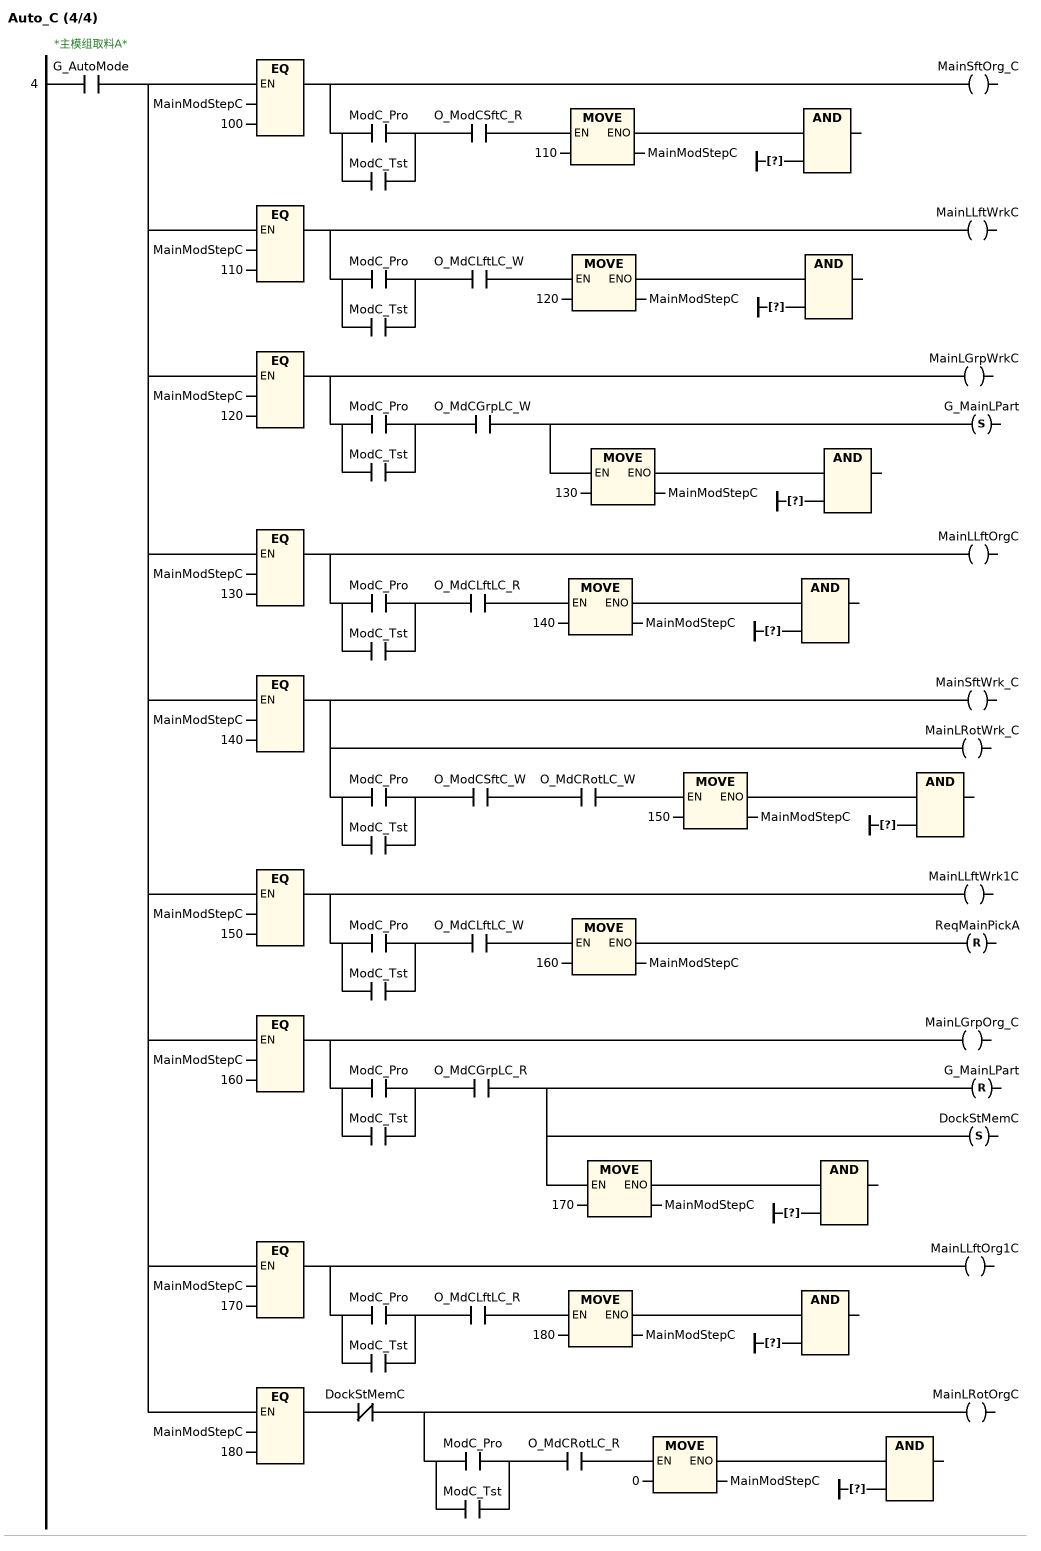
// NETWORK 4
// *主模组取料A*
_w22 := G_AutoMode AND MainModStepC = 100;
MainSftOrg_C := _w22;
_w23 := (_w22 AND ModC_Pro OR _w22 AND ModC_Tst) AND O_ModCSftC_R;
IF _w23 THEN MainModStepC := 110; END_IF
_w24 := G_AutoMode AND MainModStepC = 110;
MainLLftWrkC := _w24;
_w25 := (_w24 AND ModC_Pro OR _w24 AND ModC_Tst) AND O_MdCLftLC_W;
IF _w25 THEN MainModStepC := 120; END_IF
_w26 := G_AutoMode AND MainModStepC = 120;
MainLGrpWrkC := _w26;
_w27 := (_w26 AND ModC_Pro OR _w26 AND ModC_Tst) AND O_MdCGrpLC_W;
G_MainLPart S= _w27;
IF _w27 THEN MainModStepC := 130; END_IF
_w28 := G_AutoMode AND MainModStepC = 130;
MainLLftOrgC := _w28;
_w29 := (_w28 AND ModC_Pro OR _w28 AND ModC_Tst) AND O_MdCLftLC_R;
IF _w29 THEN MainModStepC := 140; END_IF
_w30 := G_AutoMode AND MainModStepC = 140;
MainSftWrk_C := _w30;
MainLRotWrk_C := _w30;
_w31 := (_w30 AND ModC_Pro OR _w30 AND ModC_Tst) AND O_ModCSftC_W AND O_MdCRotLC_W;
IF _w31 THEN MainModStepC := 150; END_IF
_w32 := G_AutoMode AND MainModStepC = 150;
MainLLftWrk1C := _w32;
_w33 := (_w32 AND ModC_Pro OR _w32 AND ModC_Tst) AND O_MdCLftLC_W;
IF _w33 THEN MainModStepC := 160; END_IF
ReqMainPickA R= _w33;
_w34 := G_AutoMode AND MainModStepC = 160;
MainLGrpOrg_C := _w34;
_w35 := (_w34 AND ModC_Pro OR _w34 AND ModC_Tst) AND O_MdCGrpLC_R;
G_MainLPart R= _w35;
DockStMemC S= _w35;
IF _w35 THEN MainModStepC := 170; END_IF
_w36 := G_AutoMode AND MainModStepC = 170;
MainLLftOrg1C := _w36;
_w37 := (_w36 AND ModC_Pro OR _w36 AND ModC_Tst) AND O_MdCLftLC_R;
IF _w37 THEN MainModStepC := 180; END_IF
_w38 := (G_AutoMode AND MainModStepC = 180) AND NOT DockStMemC;
MainLRotOrgC := _w38;
_w39 := (_w38 AND ModC_Pro OR _w38 AND ModC_Tst) AND O_MdCRotLC_R;
IF _w39 THEN MainModStepC := 0; END_IF

END_PROGRAM

// Device/Application/03_程序/输出/Cylinder_AZone
PROGRAM Cylinder_AZone
VAR
	StopA1Hm :BOOL;
	StopA1Wk :BOOL;
	StopA2Hm :BOOL;
	StopA2Wk :BOOL;
	StopA3Hm :BOOL;
	StopA3Wk :BOOL;
	StopA4Hm :BOOL;
	StopA4Wk :BOOL;
	StopA5Hm :BOOL;
	StopA5Wk :BOOL;
	LiftA1Hm: BOOL;
	LiftA1Wk: BOOL ;
	LiftA2Hm: BOOL;
	LiftA2Wk: BOOL ;
	LiftA3Hm: BOOL;
	LiftA3Wk: BOOL ;
	LiftA4Hm: BOOL;
	LiftA4Wk: BOOL ;
	SwtchA1Hm: BOOL;
	SwtchA1Wk: BOOL ;
	ModTrvAHm: BOOL;
	ModTrvAWk: BOOL ;
	ModClpAHm: BOOL;
	ModClpAWk: BOOL; 
	ModRotAHm: BOOL;
	ModRotAWk: BOOL; 
	
	FB_StopA1: FB_Cylinder;
	FB_StopA2: FB_Cylinder;
	FB_StopA3: FB_Cylinder;
	FB_StopA4: FB_Cylinder;
	FB_StopA5: FB_Cylinder;
	FB_LiftA1: FB_Cylinder;
    FB_LiftA2: FB_Cylinder;
    FB_LiftA3: FB_Cylinder;
    FB_LiftA4: FB_Cylinder;
	FB_SwtchA1: FB_Cylinder;
	FB_ModTrvA: FB_Cylinder;
	FB_ModClpA: FB_Cylinder;
	FB_ModRotA: FB_Cylinder;
END_VAR

//阻挡气缸A1//
IF (G_ManMode AND H_StpC_R_A1) OR LnCylInit_A.Y_BlkCylR1 OR St1Org_A
THEN StopA1Hm:=TRUE;
ELSE StopA1Hm:=FALSE;
END_IF;
IF (G_ManMode AND H_StpC_W_A1) OR St1Work_A
THEN StopA1Wk:=TRUE;
ELSE StopA1Wk:=FALSE;
END_IF;
FB_StopA1(
 X_EN:=1,
 X_HomeInBit:=X_StpCyl_R_A1,
 X_WorkInBit:=X_StpCyl_W_A1,
 X_HomeCmdBit:=StopA1Hm,
 X_WorkCmdBit:=StopA1Wk,
 X_HomeMskBit:=H_StpCR_A1_M,
 X_WorkMskBit:=H_StpCW_A1_M,
 X_HomeConfT:=H_StpCRPosDyA1,
 X_WorkConfT:=H_StpCWPosDyA1,
 X_TimeoutSet:=H_StpCTO_DlyA1,
 X_HomeMskDly:=H_StpCRMaskDyA1,
 X_WorkMskDly:=H_StpCWMaskDyA1,
 Y_ENO=>,
 Y_AtHome=>O_StpC_R_A1,
 Y_AtWork=>O_StpC_W_A1,
 Y_HomeTout=>O_StpCRFltA1,
 Y_WorkTout=>O_StpCRFltA1,
 Y_HomeOutBit=>Q_StpCyl_R_A1,
 Y_WorkOutBit=>Q_StpCyl_W_A1);
//阻挡气缸A2//
IF (G_ManMode AND H_StpC_R_A2) OR LnCylInit_A.Y_BlkCylR2 OR St2Org_A
THEN StopA2Hm:=TRUE;
ELSE StopA2Hm:=FALSE;
END_IF;
IF (G_ManMode AND H_StpC_W_A2)  OR St2Work_A
THEN StopA2Wk:=TRUE;
ELSE StopA2Wk:=FALSE;
END_IF;
FB_StopA2(
 X_EN:=1,
 X_HomeInBit:=X_StpCyl_R_A2,
 X_WorkInBit:=X_StpCyl_W_A2,
 X_HomeCmdBit:=StopA2Hm,
 X_WorkCmdBit:=StopA2Wk,
 X_HomeMskBit:=H_StpCR_A2_M,
 X_WorkMskBit:=H_StpCW_A2_M,
 X_HomeConfT:=H_StpCRPosDyA2,
 X_WorkConfT:=H_StpCWPosDyA2,
 X_TimeoutSet:=H_StpCTO_DlyA2,
 X_HomeMskDly:=H_StpCRMaskDyA2,
 X_WorkMskDly:=H_StpCWMaskDyA2,
 Y_ENO=>,
 Y_AtHome=>O_StpC_R_A2,
 Y_AtWork=>O_StpC_W_A2,
 Y_HomeTout=>O_StpCRFltA2,
 Y_WorkTout=>O_StpCWFltA2,
 Y_HomeOutBit=>Q_StpCyl_R_A2,
 Y_WorkOutBit=>Q_StpCyl_W_A2);
//阻挡气缸A3//
IF (G_ManMode AND H_StpC_R_A3) OR LnCylInit_A.Y_BlkCylR3 OR St3Org_A
THEN StopA3Hm:=TRUE;
ELSE StopA3Hm:=FALSE;
END_IF;
IF (G_ManMode AND H_StpC_W_A3)  OR St3Work_A OR St3Work1_A
THEN StopA3Wk:=TRUE;
ELSE StopA3Wk:=FALSE;
END_IF;
FB_StopA3(
 X_EN:=1,
 X_HomeInBit:=X_StpCyl_R_A3,
 X_WorkInBit:=X_StpCyl_W_A3,
 X_HomeCmdBit:=StopA3Hm,
 X_WorkCmdBit:=StopA3Wk,
 X_HomeMskBit:=H_StpCR_A3_M,
 X_WorkMskBit:=H_StpCW_A3_M,
 X_HomeConfT:=H_StpCRPosDyA3,
 X_WorkConfT:=H_StpCWPosDyA3,
 X_TimeoutSet:=H_StpCTO_DlyA3,
 X_HomeMskDly:=H_StpCRMaskDyA3,
 X_WorkMskDly:=H_StpCWMaskDyA3,
 Y_ENO=>,
 Y_AtHome=>O_StpC_R_A3,
 Y_AtWork=>O_StpC_W_A3,
 Y_HomeTout=>O_StpCRFltA3,
 Y_WorkTout=>O_StpCWFltA3,
 Y_HomeOutBit=>Q_StpCyl_R_A3,
 Y_WorkOutBit=>Q_StpCyl_W_A3);
//阻挡气缸A4//
IF (G_ManMode AND H_StpC_R_A4) OR LnCylInit_A.Y_BlkCylR4 OR St4Org_A
THEN StopA4Hm:=TRUE;
ELSE StopA4Hm:=FALSE;
END_IF;
IF (G_ManMode AND H_StpC_W_A4)  OR St4Work_A
THEN StopA4Wk:=TRUE;
ELSE StopA4Wk:=FALSE;
END_IF;
FB_StopA4(
 X_EN:=1,
 X_HomeInBit:=X_StpCyl_R_A4,
 X_WorkInBit:=X_StpCyl_W_A4,
 X_HomeCmdBit:=StopA4Hm,
 X_WorkCmdBit:=StopA4Wk,
 X_HomeMskBit:=H_StpCR_A4_M,
 X_WorkMskBit:=H_StpCW_A4_M,
 X_HomeConfT:=H_StpCRPosDyA4,
 X_WorkConfT:=H_StpCWPosDyA4,
 X_TimeoutSet:=H_StpCTO_DlyA4,
 X_HomeMskDly:=H_StpCRMaskDyA4,
 X_WorkMskDly:=H_StpCWMaskDyA4,
 Y_ENO=>,
 Y_AtHome=>O_StpC_R_A4,
 Y_AtWork=>O_StpC_W_A4,
 Y_HomeTout=>O_StpCRFltA4,
 Y_WorkTout=>O_StpCWFltA4,
 Y_HomeOutBit=>Q_StpCyl_R_A4,
 Y_WorkOutBit=>Q_StpCyl_W_A4);
//阻挡气缸A5//
IF (G_ManMode AND H_StpC_R_A5) OR LnCylInit_A.Y_BlkCylR5 OR St5Org_A
THEN StopA5Hm:=TRUE;
ELSE StopA5Hm:=FALSE;
END_IF;
IF (G_ManMode AND H_StpC_W_A5) OR St5Work_A
THEN StopA5Wk:=TRUE;
ELSE StopA5Wk:=FALSE;
END_IF;
FB_StopA5(
 X_EN:=1,
 X_HomeInBit:=X_StpCyl_R_A5,
 X_WorkInBit:=X_StpCyl_W_A5,
 X_HomeCmdBit:=StopA5Hm,
 X_WorkCmdBit:=StopA5Wk,
 X_HomeMskBit:=H_StpCR_A5_M,
 X_WorkMskBit:=H_StpCW_A5_M,
 X_HomeConfT:=H_StpCRPosDyA5,
 X_WorkConfT:=H_StpCWPosDyA5,
 X_TimeoutSet:=H_StpCTO_DlyA5,
 X_HomeMskDly:=H_StpCRMaskDyA5,
 X_WorkMskDly:=H_StpCWMaskDyA5,
 Y_ENO=>,
 Y_AtHome=>O_StpC_R_A5,
 Y_AtWork=>O_StpC_W_A5,
 Y_HomeTout=>O_StpCRFltA5,
 Y_WorkTout=>O_StpCWFltA5,
 Y_HomeOutBit=>Q_StpCyl_R_A5,
 Y_WorkOutBit=>Q_StpCyl_W_A5);
//顶升气缸A1//
IF (G_ManMode AND H_LftC_R_A1) OR LnCylInit_A.Y_LftCylR1 OR UD1Org_A OR UD1OrgPos1_A
THEN LiftA1Hm:=TRUE;
ELSE LiftA1Hm:=FALSE;
END_IF;
IF (G_ManMode AND H_LftC_W_A1) OR LnCylInit_A.Y_LftCylM1 OR UD1Work_A OR UD1Work1_A
THEN LiftA1Wk:=TRUE;
ELSE LiftA1Wk:=FALSE;
END_IF;
FB_LiftA1(
 X_EN:=1,
 X_HomeInBit:=X_LftCyl_R_A1,
 X_WorkInBit:=X_LftCyl_W_A1,
 X_HomeCmdBit:=LiftA1Hm,
 X_WorkCmdBit:=LiftA1Wk,
 X_HomeMskBit:=H_LftCR_A1_M,
 X_WorkMskBit:=H_LftCW_A1_M,
 X_HomeConfT:=H_LftCRPosDyA1,
 X_WorkConfT:=H_LftCWPosDyA1,
 X_TimeoutSet:=H_LftCTO_DlyA1,
 X_HomeMskDly:=H_LftCRMaskDyA1,
 X_WorkMskDly:=H_LftCWMaskDyA1,
 Y_ENO=>,
 Y_AtHome=>O_LftC_R_A1,
 Y_AtWork=>O_LftC_W_A1,
 Y_HomeTout=>O_LftCRFltA1,
 Y_WorkTout=>O_LftCWFltA1,
 Y_HomeOutBit=>Q_LftCyl_R_A1,
 Y_WorkOutBit=>Q_LftCyl_W_A1);
//顶升气缸A2//
IF (G_ManMode AND H_LftC_R_A2) OR LnCylInit_A.Y_LftCylR2 OR UD2Org_A
THEN LiftA2Hm:=TRUE;
ELSE LiftA2Hm:=FALSE;
END_IF;
IF (G_ManMode AND H_LftC_W_A2)  OR UD2Work_A
THEN LiftA2Wk:=TRUE;
ELSE LiftA2Wk:=FALSE;
END_IF;
FB_LiftA2(
 X_EN:=1,
 X_HomeInBit:=X_LftCyl_R_A2,
 X_WorkInBit:=X_LftCyl_W_A2,
 X_HomeCmdBit:=LiftA2Hm,
 X_WorkCmdBit:=LiftA2Wk,
 X_HomeMskBit:=H_LftCR_A2_M,
 X_WorkMskBit:=H_LftCW_A2_M,
 X_HomeConfT:=H_LftCRPosDyA2,
 X_WorkConfT:=H_LftCWPosDyA2,
 X_TimeoutSet:=H_LftCTO_DlyA2,
 X_HomeMskDly:=H_LftCRMaskDyA2,
 X_WorkMskDly:=H_LftCWMaskDyA2,
 Y_ENO=>,
 Y_AtHome=>O_LftC_R_A2,
 Y_AtWork=>O_LftC_W_A2,
 Y_HomeTout=>O_LftCRFltA2,
 Y_WorkTout=>O_LftCWFltA2,
 Y_HomeOutBit=>Q_LftCyl_R_A2,
 Y_WorkOutBit=>Q_LftCyl_W_A2);
//顶升气缸A3//
IF (G_ManMode AND H_LftC_R_A3) OR LnCylInit_A.Y_LftCylR3 OR UD3Org_A
THEN LiftA3Hm:=TRUE;
ELSE LiftA3Hm:=FALSE;
END_IF;
IF (G_ManMode AND H_LftC_W_A3)  OR UD3Work_A
THEN LiftA3Wk:=TRUE;
ELSE LiftA3Wk:=FALSE;
END_IF;
FB_LiftA3(
 X_EN:=1,
 X_HomeInBit:=X_LftCyl_R_A3,
 X_WorkInBit:=X_LftCyl_W_A3,
 X_HomeCmdBit:=LiftA3Hm,
 X_WorkCmdBit:=LiftA3Wk,
 X_HomeMskBit:=H_LftCR_A3_M,
 X_WorkMskBit:=H_LftCW_A3_M,
 X_HomeConfT:=H_LftCRPosDyA3,
 X_WorkConfT:=H_LftCWPosDyA3,
 X_TimeoutSet:=H_LftCTO_DlyA3,
 X_HomeMskDly:=H_LftCRMaskDyA3,
 X_WorkMskDly:=H_LftCWMaskDyA3,
 Y_ENO=>,
 Y_AtHome=>O_LftC_R_A3,
 Y_AtWork=>O_LftC_W_A3,
 Y_HomeTout=>O_LftCRFltA3,
 Y_WorkTout=>O_LftCWFltA3,
 Y_HomeOutBit=>Q_LftCyl_R_A3,
 Y_WorkOutBit=>Q_LftCyl_W_A3);
//顶升气缸A4//
IF (G_ManMode AND H_LftC_R_A4) OR LnCylInit_A.Y_LftCylR4 OR UD4Org_A
THEN LiftA4Hm:=TRUE;
ELSE LiftA4Hm:=FALSE;
END_IF;
IF (G_ManMode AND H_LftC_W_A4)  OR UD4Work_A
THEN LiftA4Wk:=TRUE;
ELSE LiftA4Wk:=FALSE;
END_IF;
FB_LiftA4(
 X_EN:=1,
 X_HomeInBit:=X_LftCyl_R_A4,
 X_WorkInBit:=X_LftCyl_W_A4,
 X_HomeCmdBit:=LiftA4Hm,
 X_WorkCmdBit:=LiftA4Wk,
 X_HomeMskBit:=H_LftCR_A4_M,
 X_WorkMskBit:=H_LftCW_A4_M,
 X_HomeConfT:=H_LftCRPosDyA4,
 X_WorkConfT:=H_LftCWPosDyA4,
 X_TimeoutSet:=H_LftCTO_DlyA4,
 X_HomeMskDly:=H_LftCRMaskDyA4,
 X_WorkMskDly:=H_LftCWMaskDyA4,
 Y_ENO=>,
 Y_AtHome=>O_LftC_R_A4,
 Y_AtWork=>O_LftC_W_A4,
 Y_HomeTout=>O_LftCRFltA4,
 Y_WorkTout=>O_LftCWFltA4,
 Y_HomeOutBit=>Q_LftCyl_R_A4,
 Y_WorkOutBit=>Q_LftCyl_W_A4);
//换向气缸A1//
IF (G_ManMode AND H_TrnC_R_A1 AND O_LftC_W_A1) OR LnCylInit_A.Y_StrCylO1 OR RevOrg_A
THEN SwtchA1Hm:=TRUE;
ELSE SwtchA1Hm:=FALSE;
END_IF;
IF (G_ManMode AND H_TrnC_W_A1 AND O_LftC_W_A1)  OR RevWork_A
THEN SwtchA1Wk:=TRUE;
ELSE SwtchA1Wk:=FALSE;
END_IF;
FB_SwtchA1(
 X_EN:=1,
 X_HomeInBit:=X_TrnCyl_R_A1,
 X_WorkInBit:=X_TrnCyl_W_A1,
 X_HomeCmdBit:=SwtchA1Hm,
 X_WorkCmdBit:=SwtchA1Wk,
 X_HomeMskBit:=H_TrnCR_A1_M,
 X_WorkMskBit:=H_TrnCW_A1_M ,
 X_HomeConfT:=H_TrnCRPosDyA1,
 X_WorkConfT:=H_TrnCWPosDyA1,
 X_TimeoutSet:=H_TrnCTO_DlyA1,
 X_HomeMskDly:=H_TrnCRMaskDyA1,
 X_WorkMskDly:=H_TrnCWMaskDyA1,
 Y_ENO=>,
 Y_AtHome=>O_TrnC_R_A1,
 Y_AtWork=>O_TrnC_W_A1,
 Y_HomeTout=>O_TrnCRFltA1,
 Y_WorkTout=>O_TrnCWFltA1,
 Y_HomeOutBit=>Q_TrnCyl_R_A1,
 Y_WorkOutBit=>Q_TrnCyl_W_A1);
//模组平移气缸A//
IF (G_ManMode AND H_ModASftC_R AND Ax1GoP1) OR PickModInitA.Y_TrnCylR OR SftCylOrg_A
THEN ModTrvAHm:=TRUE;
ELSE ModTrvAHm:=FALSE;
END_IF;
IF (G_ManMode AND H_ModASftC_W AND Ax1GoP1)  OR SftCylWork_A
THEN ModTrvAWk:=TRUE;
ELSE ModTrvAWk:=FALSE;
END_IF;
FB_ModTrvA(
 X_EN:=1,
 X_HomeInBit:=X_ModASftC_R,
 X_WorkInBit:=X_ModASftC_W,
 X_HomeCmdBit:=ModTrvAHm,
 X_WorkCmdBit:=ModTrvAWk,
 X_HomeMskBit:=H_MdASftCR_M,
 X_WorkMskBit:=H_MdASftCW_M,
 X_HomeConfT:=H_MASftCRPosDy,
 X_WorkConfT:=H_MASftCWPosDy,
 X_TimeoutSet:=H_MASftCTO_Dly,
 X_HomeMskDly:=H_MASftCRMaskDy,
 X_WorkMskDly:=H_MASftCWMaskDy,
 Y_ENO=>,
 Y_AtHome=>O_ModASftC_R,
 Y_AtWork=>O_ModASftC_W,
 Y_HomeTout=>O_MASftCRFlt,
 Y_WorkTout=>O_MASftCWFlt,
 Y_HomeOutBit=>Q_ModASftC_R,
 Y_WorkOutBit=>Q_ModASftC_W);
//模组夹取气缸A//
IF (G_ManMode AND H_ModAGrpC_R) OR PickModInitA.Y_ClmpCylO OR GripCylOrg_A
THEN ModClpAHm:=TRUE;
ELSE ModClpAHm:=FALSE;
END_IF;
IF (G_ManMode AND H_ModAGrpC_W) OR GripCylWorkA
THEN ModClpAWk:=TRUE;
ELSE ModClpAWk:=FALSE;
END_IF;
FB_ModClpA(
 X_EN:=1,
 X_HomeInBit:=X_ModAGrpC_R,
 X_WorkInBit:=X_ModAGrpC_W,
 X_HomeCmdBit:=ModClpAHm,
 X_WorkCmdBit:=ModClpAWk,
 X_HomeMskBit:=H_MdAGrpCR_M,
 X_WorkMskBit:=H_MdAGrpCW_M,
 X_HomeConfT:=H_MAGrpCRPosDy,
 X_WorkConfT:=H_MAGrpCWPosDy,
 X_TimeoutSet:=H_MAGrpCTO_Dly,
 X_HomeMskDly:=H_MAGrpCRMaskDy,
 X_WorkMskDly:=H_MAGrpCWMaskDy,
 Y_ENO=>,
 Y_AtHome=>O_ModAGrpC_R,
 Y_AtWork=>O_ModAGrpC_W,
 Y_HomeTout=>O_MAGrpCRFlt,
 Y_WorkTout=>O_MAGrpCWFlt,
 Y_HomeOutBit=>Q_ModAGrpC_R,
 Y_WorkOutBit=>Q_ModAGrpC_W);
//模组旋转气缸A//
IF (G_ManMode AND H_ModARotC_R) OR PickModInitA.Y_RotCylO OR RotCylOrg_A
THEN ModRotAHm:=TRUE;
ELSE ModRotAHm:=FALSE;
END_IF;
IF (G_ManMode AND H_ModARotC_W) OR RotCylWork_A
THEN ModRotAWk:=TRUE;
ELSE ModRotAWk:=FALSE;
END_IF;
FB_ModRotA(
 X_EN:=1,
 X_HomeInBit:=X_ModARotC_R,
 X_WorkInBit:=X_ModARotC_W,
 X_HomeCmdBit:=ModRotAHm,
 X_WorkCmdBit:=ModRotAWk,
 X_HomeMskBit:=H_MdARotCR_M,
 X_WorkMskBit:=H_MdARotCW_M,
 X_HomeConfT:=H_MARotCRPosDy,
 X_WorkConfT:=H_MARotCWPosDy,
 X_TimeoutSet:=H_MARotCTO_Dly,
 X_HomeMskDly:=H_MARotCRMaskDy,
 X_WorkMskDly:=H_MARotCWMaskDy,
 Y_ENO=>,
 Y_AtHome=>O_ModARotC_R,
 Y_AtWork=>O_ModARotC_W,
 Y_HomeTout=>O_MARotCRFlt,
 Y_WorkTout=>O_MARotCWFlt,
 Y_HomeOutBit=>Q_ModARotC_R,
 Y_WorkOutBit=>Q_ModARotC_W);

END_PROGRAM

// Device/Application/02_功能块/气缸/FB_Cylinder
FUNCTION_BLOCK FB_Cylinder
VAR_INPUT
	X_EN: BOOL;
	X_HomeInBit: BOOL;
	X_WorkInBit: BOOL;
	X_HomeCmdBit: BOOL;
	X_WorkCmdBit: BOOL;
	X_HomeMskBit: BOOL;
	X_WorkMskBit: BOOL;
	X_HomeConfT: TIME;
	X_WorkConfT: TIME;
	X_TimeoutSet: TIME;
	X_HomeMskDly: TIME;
	X_WorkMskDly: TIME;
END_VAR
VAR_OUTPUT
	Y_ENO: BOOL;
	Y_AtHome: BOOL;
	Y_AtWork: BOOL;
	Y_HomeTout: BOOL;
	Y_WorkTout: BOOL;
	Y_HomeOutBit: BOOL;
	Y_WorkOutBit: BOOL;	
END_VAR
VAR
	TON_0: TON;
	TON_1: TON;
	TON_2: TON;
	TON_3: TON;
	TON_4: TON;
	TON_5: TON;
	R_TRIG_0: R_TRIG;
	END_VAR
VAR // added by the converter: edge detectors and wires of the graphical bodies
    _w1, _w2, _w3, _w4, _w5 : BOOL;
END_VAR

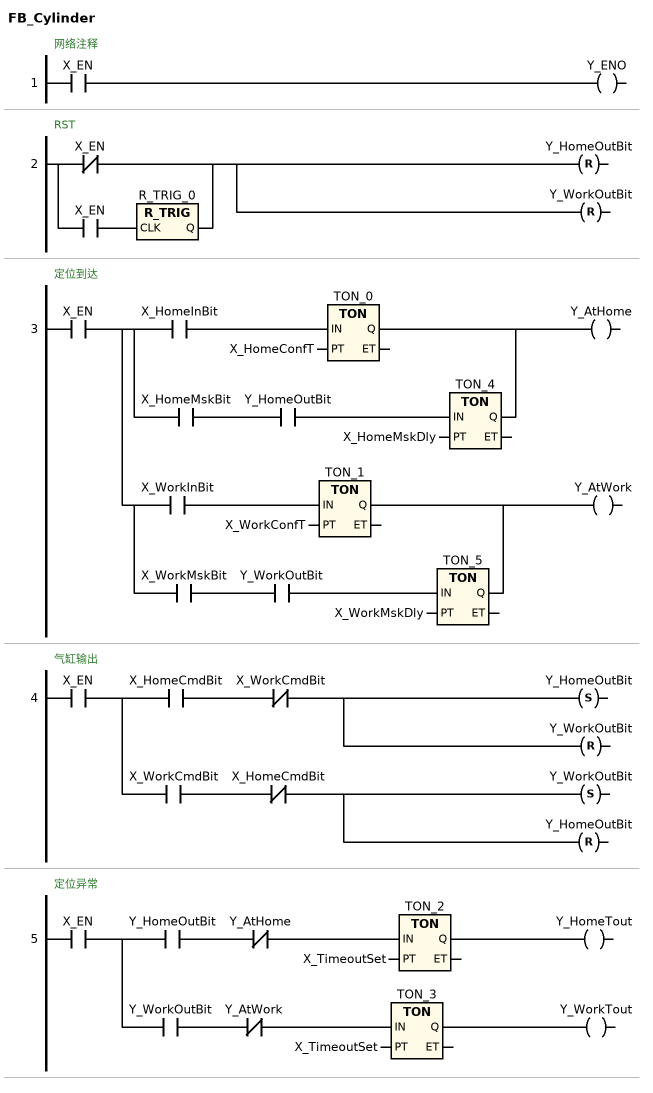
// NETWORK 1
// 网络注释
Y_ENO := X_EN;

// NETWORK 2
// RST
R_TRIG_0(CLK := X_EN); // R_TRIG
_w1 := NOT X_EN OR R_TRIG_0.Q;
Y_HomeOutBit R= _w1;
Y_WorkOutBit R= _w1;

// NETWORK 3
// 定位到达
TON_0(IN := X_EN AND X_HomeInBit, PT := X_HomeConfT); // TON
TON_4(IN := (X_EN AND X_HomeMskBit) AND Y_HomeOutBit, PT := X_HomeMskDly); // TON
_w2 := TON_0.Q OR TON_4.Q;
Y_AtHome := _w2;
TON_1(IN := X_EN AND X_WorkInBit, PT := X_WorkConfT); // TON
TON_5(IN := (X_EN AND X_WorkMskBit) AND Y_WorkOutBit, PT := X_WorkMskDly); // TON
_w3 := TON_1.Q OR TON_5.Q;
Y_AtWork := _w3;

// NETWORK 4
// 气缸输出
_w4 := (X_EN AND X_HomeCmdBit) AND NOT X_WorkCmdBit;
Y_HomeOutBit S= _w4;
Y_WorkOutBit R= _w4;
_w5 := (X_EN AND X_WorkCmdBit) AND NOT X_HomeCmdBit;
Y_WorkOutBit S= _w5;
Y_HomeOutBit R= _w5;

// NETWORK 5
// 定位异常
TON_2(IN := (X_EN AND Y_HomeOutBit) AND NOT Y_AtHome, PT := X_TimeoutSet); // TON
Y_HomeTout := TON_2.Q;
TON_3(IN := (X_EN AND Y_WorkOutBit) AND NOT Y_AtWork, PT := X_TimeoutSet); // TON
Y_WorkTout := TON_3.Q;

END_FUNCTION_BLOCK

// Device/Application/03_程序/输出/Cylinder_CZone
PROGRAM Cylinder_CZone
VAR
 StopC1Hm :BOOL;
 StopC1Wk :BOOL;
 LiftC1Hm: BOOL;
 LiftC1Wk: BOOL ;
ModTrvCHm :BOOL;
ModTrvCWk :BOOL;
ModLLftCHm :BOOL;
ModLLftCWk :BOOL;
ModLClpCHm :BOOL;
ModLClpCWk :BOOL;
ModLRotCHm :BOOL;
ModLRotCWk :BOOL;

 
 FB_StopC1: FB_Cylinder;
 FB_LiftC1: FB_Cylinder;
 FB_ModTrvC: FB_Cylinder;
 FB_ModLLftC: FB_Cylinder;
 FB_ModLClpC: FB_Cylinder;
 FB_ModLRotC: FB_Cylinder;
END_VAR

//阻挡气缸C1//
IF (G_ManMode AND H_StpC_R_C1) OR DockCylInitC.Y_BlkCylR OR StpCylOrg_C
THEN StopC1Hm:=TRUE;
ELSE StopC1Hm:=FALSE;
END_IF;
IF (G_ManMode AND H_StpC_W_C1) OR StpCylWork_C
THEN StopC1Wk:=TRUE;
ELSE StopC1Wk:=FALSE;
END_IF;
FB_StopC1(
 X_EN:=1,
 X_HomeInBit:=X_StpCyl_R_C1,
 X_WorkInBit:=X_StpCyl_W_C1,
 X_HomeCmdBit:=StopC1Hm,
 X_WorkCmdBit:=StopC1Wk,
 X_HomeMskBit:=H_StpCR_C1_M,
 X_WorkMskBit:=H_StpCW_C1_M,
 X_HomeConfT:=H_StpCRPosDyC1,
 X_WorkConfT:=H_StpCWPosDyC1,
 X_TimeoutSet:=H_StpCTO_DlyC1,
 X_HomeMskDly:=H_StpCRMaskDyC1,
 X_WorkMskDly:=H_StpCWMaskDyC1,
 Y_ENO=>,
 Y_AtHome=>O_StpC_R_C1,
 Y_AtWork=>O_StpC_W_C1,
 Y_HomeTout=>O_StpCRFltC1,
 Y_WorkTout=>O_StpCWFltC1,
 Y_HomeOutBit=>Q_StpCyl_R_C1,
 Y_WorkOutBit=>Q_StpCyl_W_C1);
//顶升气缸C1//
IF (G_ManMode AND H_LftC_R_C1) OR DockCylInitC.Y_LftCylR OR LftCylOrg_C
THEN LiftC1Hm:=TRUE;
ELSE LiftC1Hm:=FALSE;
END_IF;
IF (G_ManMode AND H_LftC_W_C1) OR LftCylWork_C
THEN LiftC1Wk:=TRUE;
ELSE LiftC1Wk:=FALSE;
END_IF;
FB_LiftC1(
 X_EN:=1,
 X_HomeInBit:=X_LftCyl_R_C1,
 X_WorkInBit:=X_LftCyl_W_C1,
 X_HomeCmdBit:=LiftC1Hm,
 X_WorkCmdBit:=LiftC1Wk,
 X_HomeMskBit:=H_LftCR_C1_M,
 X_WorkMskBit:=H_LftCW_C1_M,
 X_HomeConfT:=H_LftCRPosDyC1,
 X_WorkConfT:=H_LftCWPosDyC1,
 X_TimeoutSet:=H_LftCTO_DlyC1,
 X_HomeMskDly:=H_LftCRMaskDyC1,
 X_WorkMskDly:=H_LftCWMaskDyC1,
 Y_ENO=>,
 Y_AtHome=>O_LftC_R_C1,
 Y_AtWork=>O_LftC_W_C1,
 Y_HomeTout=>O_LftCRFltC1,
 Y_WorkTout=>O_LftCWFltC1,
 Y_HomeOutBit=>Q_LftCyl_R_C1,
 Y_WorkOutBit=>Q_LftCyl_W_C1);
//模组平移气缸C//
IF (G_ManMode AND H_ModCSftC_R AND O_MdCLftLC_R) OR MainModInitC.Y_TrnCylR OR MainSftOrg_C OR MainSftOrg1C
THEN ModTrvCHm:=TRUE;
ELSE ModTrvCHm:=FALSE;
END_IF;
IF (G_ManMode AND H_ModCSftC_W AND O_MdCLftLC_R)  OR MainSftWrk_C OR MainSftWrk1_C
THEN ModTrvCWk:=TRUE;
ELSE ModTrvCWk:=FALSE;
END_IF;
FB_ModTrvC(
 X_EN:=1,
 X_HomeInBit:=X_ModCSftC_R,
 X_WorkInBit:=X_ModCSftC_W,
 X_HomeCmdBit:=ModTrvCHm,
 X_WorkCmdBit:=ModTrvCWk,
 X_HomeMskBit:=H_MdCSftCR_M,
 X_WorkMskBit:=H_MdCSftCW_M,
 X_HomeConfT:=H_MCSftCRPosDy,
 X_WorkConfT:=H_MCSftCWPosDy,
 X_TimeoutSet:=H_MCSftCTO_Dly,
 X_HomeMskDly:=H_MCSftCRMaskDy,
 X_WorkMskDly:=H_MCSftCWMaskDy,
 Y_ENO=>,
 Y_AtHome=>O_ModCSftC_R,
 Y_AtWork=>O_ModCSftC_W,
 Y_HomeTout=>O_MCSftCRFlt,
 Y_WorkTout=>O_MCSftCWFlt,
 Y_HomeOutBit=>Q_ModCSftC_R,
 Y_WorkOutBit=>Q_ModCSftC_W);
//模组左升降气缸C//
IF (G_ManMode AND H_MdCLftLC_R) OR MainModInitC.Y_LLftCylR OR MainLLftOrgC OR MainLLftOrg1C
THEN ModLLftCHm:=TRUE;
ELSE ModLLftCHm:=FALSE;
END_IF;
IF (G_ManMode AND H_MdCLftLC_W)  OR MainLLftWrkC  OR MainLLftWrk1C
THEN ModLLftCWk:=TRUE;
ELSE ModLLftCWk:=FALSE;
END_IF;
FB_ModLLftC(
 X_EN:=1,
 X_HomeInBit:=X_MdCLftLC_R,
 X_WorkInBit:=X_MdCLftLC_W,
 X_HomeCmdBit:=ModLLftCHm,
 X_WorkCmdBit:=ModLLftCWk,
 X_HomeMskBit:=H_MdCLftLR_M,
 X_WorkMskBit:=H_MdCLftLW_M,
 X_HomeConfT:=H_MCLftLRPosDy,
 X_WorkConfT:=H_MCLftLWPosDy,
 X_TimeoutSet:=H_MCLftLTO_Dly,
 X_HomeMskDly:=H_MCLftLRMaskDy,
 X_WorkMskDly:=H_MCLftLWMaskDy,
 Y_ENO=>,
 Y_AtHome=>O_MdCLftLC_R,
 Y_AtWork=>O_MdCLftLC_W,
 Y_HomeTout=>O_MCLftLRFlt,
 Y_WorkTout=>O_MCLftLWFlt,
 Y_HomeOutBit=>Q_MdCLftLC_R,
 Y_WorkOutBit=>Q_MdCLftLC_W);
 //模组左旋转气缸C//
 IF (G_ManMode AND H_MdCRotLC_R) OR MainModInitC.Y_LRotCylR OR MainLRotOrgC
THEN ModLRotCHm:=TRUE;
ELSE ModLRotCHm:=FALSE;
END_IF;
IF (G_ManMode AND H_MdCRotLC_W)  OR MainLRotWrk_C
THEN ModLRotCWk:=TRUE;
ELSE ModLRotCWk:=FALSE;
END_IF;
FB_ModLRotC(
 X_EN:=1,
 X_HomeInBit:=X_MdCRotLC_R,
 X_WorkInBit:=X_MdCRotLC_W,
 X_HomeCmdBit:=ModLRotCHm,
 X_WorkCmdBit:=ModLRotCWk,
 X_HomeMskBit:=H_MdCRotLR_M,
 X_WorkMskBit:=H_MdCRotLW_M,
 X_HomeConfT:=H_MCRotLRPosDy,
 X_WorkConfT:=H_MCRotLWPosDy,
 X_TimeoutSet:=H_MCRotLTO_Dly,
 X_HomeMskDly:=H_MCRotLRMaskDy,
 X_WorkMskDly:=H_MCRotLWMaskDy,
 Y_ENO=>,
 Y_AtHome=>O_MdCRotLC_R,
 Y_AtWork=>O_MdCRotLC_W,
 Y_HomeTout=>O_MCRotLRFlt,
 Y_WorkTout=>O_MCRotLWFlt,
 Y_HomeOutBit=>Q_MdCRotLC_R,
 Y_WorkOutBit=>Q_MdCRotLC_W);
 //模组左夹取气缸C//
IF (G_ManMode AND H_MdCGrpLC_R) OR MainModInitC.Y_LClmpCylR OR MainLGrpOrg_C
THEN ModLClpCHm:=TRUE;
ELSE ModLClpCHm:=FALSE;
END_IF;
IF (G_ManMode AND H_MdCGrpLC_W)  OR MainLGrpWrkC 
THEN ModLClpCWk:=TRUE;
ELSE ModLClpCWk:=FALSE;
END_IF;
FB_ModLClpC(
 X_EN:=1,
 X_HomeInBit:=X_MdCGrpLC_R,
 X_WorkInBit:=X_MdCGrpLC_W,
 X_HomeCmdBit:=ModLClpCHm,
 X_WorkCmdBit:=ModLClpCWk,
 X_HomeMskBit:=H_MdCGrpLR_M,
 X_WorkMskBit:=H_MdCGrpLW_M,
 X_HomeConfT:=H_MCGrpLRPosDy,
 X_WorkConfT:=H_MCGrpLWPosDy,
 X_TimeoutSet:=H_MCGrpLTO_Dly,
 X_HomeMskDly:=H_MCGrpLRMaskDy,
 X_WorkMskDly:=H_MCGrpLWMaskDy,
 Y_ENO=>,
 Y_AtHome=>O_MdCGrpLC_R,
 Y_AtWork=>O_MdCGrpLC_W,
 Y_HomeTout=>O_MCGrpLRFlt,
 Y_WorkTout=>O_MCGrpLWFlt,
 Y_HomeOutBit=>Q_MdCGrpLC_R,
 Y_WorkOutBit=>Q_MdCGrpLC_W);

END_PROGRAM

// Device/Application/03_程序/输出/Other
PROGRAM Other
VAR	
END_VAR
VAR // added by the converter: edge detectors and wires of the graphical bodies
    _w1, _w2, _w3, _w4, _w5, _w6, _w7 : BOOL;
END_VAR

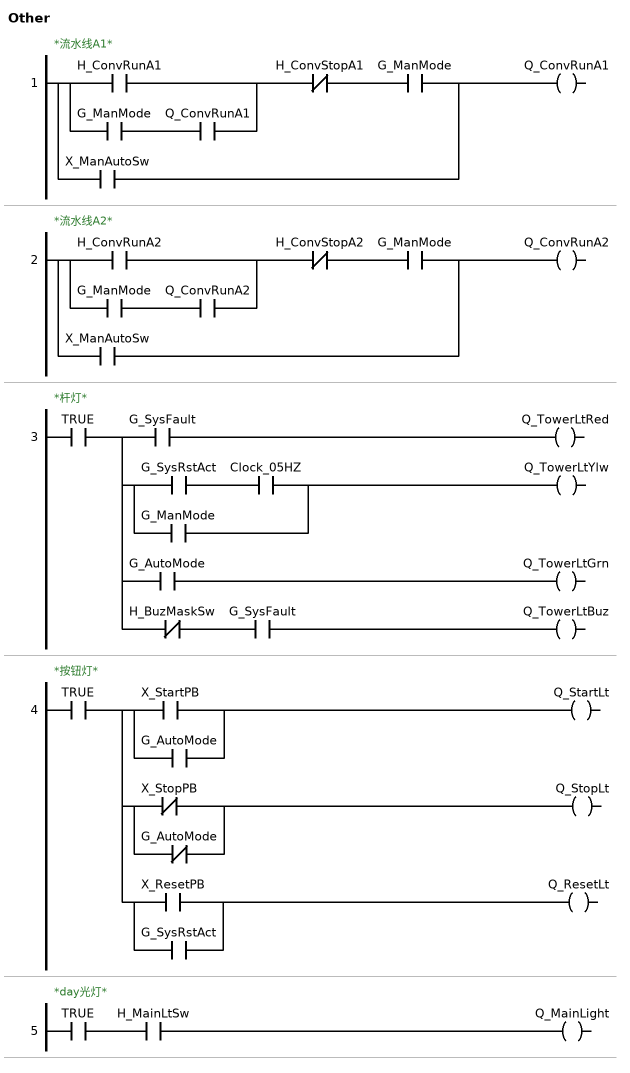
// NETWORK 1
// *流水线A1*
Q_ConvRunA1 := (H_ConvRunA1 OR G_ManMode AND Q_ConvRunA1) AND NOT H_ConvStopA1 AND G_ManMode OR X_ManAutoSw;

// NETWORK 2
// *流水线A2*
Q_ConvRunA2 := (H_ConvRunA2 OR G_ManMode AND Q_ConvRunA2) AND NOT H_ConvStopA2 AND G_ManMode OR X_ManAutoSw;

// NETWORK 3
// *杆灯*
_w1 := TRUE AND G_SysFault;
Q_TowerLtRed := _w1;
_w2 := (TRUE AND G_SysRstAct) AND Clock_05HZ OR TRUE AND G_ManMode;
Q_TowerLtYlw := _w2;
_w3 := TRUE AND G_AutoMode;
Q_TowerLtGrn := _w3;
_w4 := (TRUE AND NOT H_BuzMaskSw) AND G_SysFault;
Q_TowerLtBuz := _w4;

// NETWORK 4
// *按钮灯*
_w5 := TRUE AND X_StartPB OR TRUE AND G_AutoMode;
Q_StartLt := _w5;
_w6 := TRUE AND NOT X_StopPB OR TRUE AND NOT G_AutoMode;
Q_StopLt := _w6;
_w7 := TRUE AND X_ResetPB OR TRUE AND G_SysRstAct;
Q_ResetLt := _w7;

// NETWORK 5
// *day光灯*
Q_MainLight := TRUE AND H_MainLtSw;

END_PROGRAM

// Device/Application/03_程序/伺服控制/Axis_Teaching
PROGRAM Axis_Teaching
VAR
END_VAR
VAR // added by the converter: edge detectors and wires of the graphical bodies
    _w1, _w2, _w3, _w4, _w5 : BOOL;
END_VAR

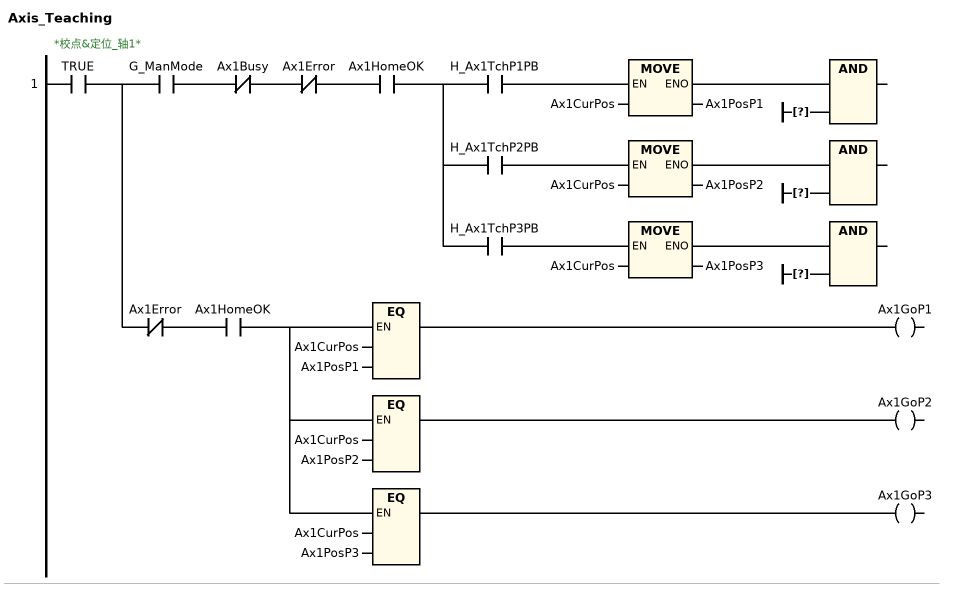
// NETWORK 1
// *校点&定位_轴1*
_w1 := (TRUE AND G_ManMode) AND NOT Ax1Busy AND NOT Ax1Error AND Ax1HomeOK;
IF _w1 AND H_Ax1TchP1PB THEN Ax1PosP1 := Ax1CurPos; END_IF
IF _w1 AND H_Ax1TchP2PB THEN Ax1PosP2 := Ax1CurPos; END_IF
IF _w1 AND H_Ax1TchP3PB THEN Ax1PosP3 := Ax1CurPos; END_IF
_w2 := (TRUE AND NOT Ax1Error) AND Ax1HomeOK;
_w3 := _w2 AND Ax1CurPos = Ax1PosP1;
Ax1GoP1 := _w3;
_w4 := _w2 AND Ax1CurPos = Ax1PosP2;
Ax1GoP2 := _w4;
_w5 := _w2 AND Ax1CurPos = Ax1PosP3;
Ax1GoP3 := _w5;

END_PROGRAM

// Device/Application/03_程序/伺服控制/Axis_Ctrl
PROGRAM Axis_Ctrl
VAR
	SerEn_1: BOOL;
	SerEn_2: BOOL;
END_VAR
VAR // added by the converter: edge detectors and wires of the graphical bodies
    _w1, _w2, _w3, _w4, _w5, _w6, _w7, _w8, _w9 : BOOL;
END_VAR

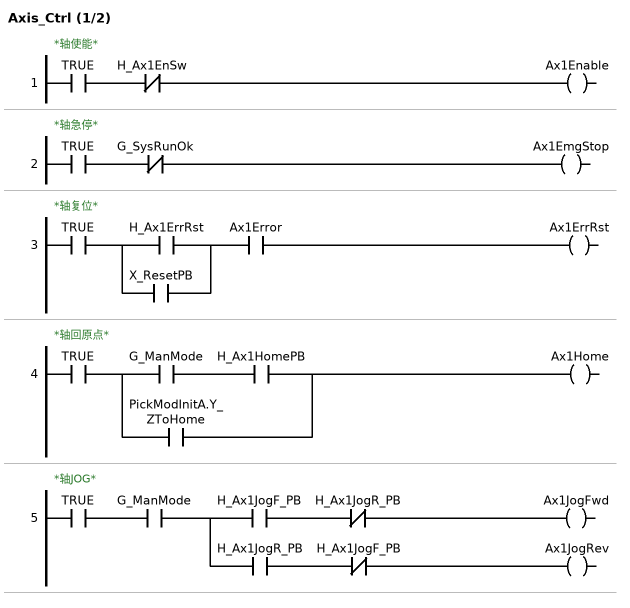
// NETWORK 1
// *轴使能*
Ax1Enable := TRUE AND NOT H_Ax1EnSw;

// NETWORK 2
// *轴急停*
Ax1EmgStop := TRUE AND NOT G_SysRunOk;

// NETWORK 3
// *轴复位*
Ax1ErrRst := (TRUE AND H_Ax1ErrRst OR TRUE AND X_ResetPB) AND Ax1Error;

// NETWORK 4
// *轴回原点*
Ax1Home := (TRUE AND G_ManMode) AND H_Ax1HomePB OR TRUE AND PickModInitA.Y_ZToHome;

// NETWORK 5
// *轴JOG*
_w1 := TRUE AND G_ManMode;
_w2 := (_w1 AND H_Ax1JogF_PB) AND NOT H_Ax1JogR_PB;
Ax1JogFwd := _w2;
_w3 := (_w1 AND H_Ax1JogR_PB) AND NOT H_Ax1JogF_PB;
Ax1JogRev := _w3;

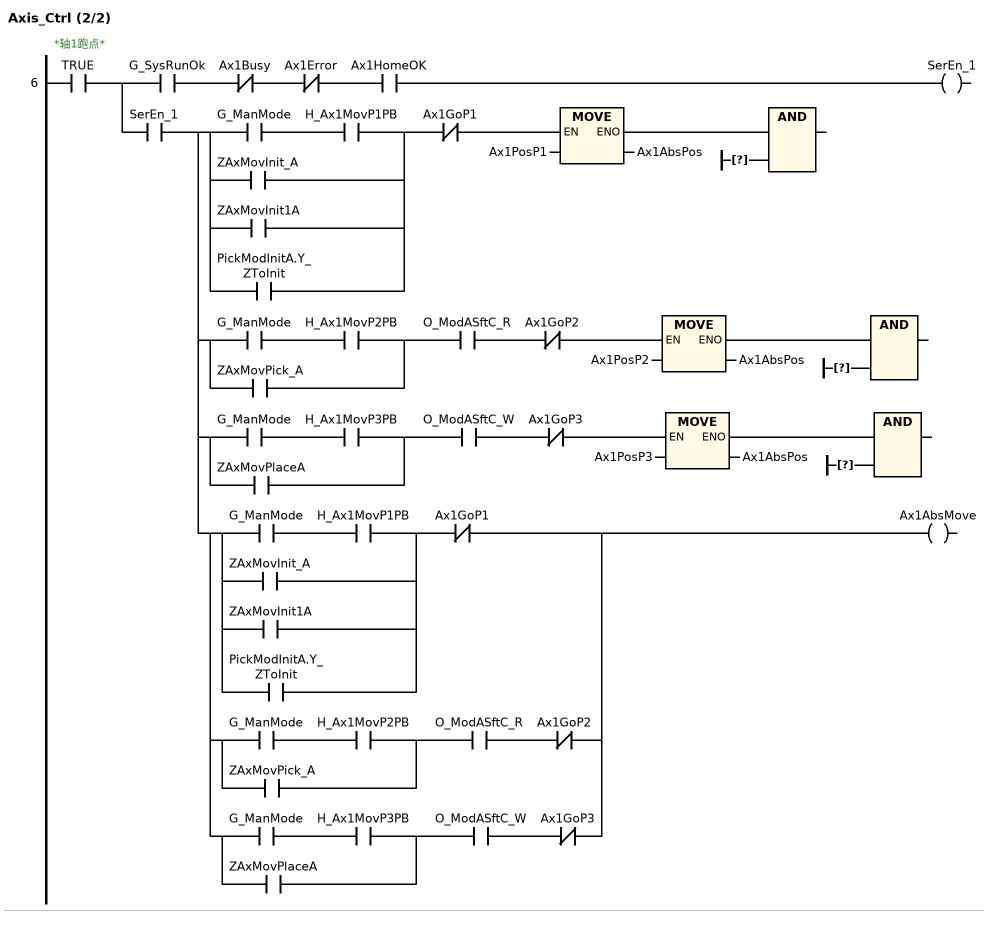
// NETWORK 6
// *轴1跑点*
_w4 := (TRUE AND G_SysRunOk) AND NOT Ax1Busy AND NOT Ax1Error AND Ax1HomeOK;
SerEn_1 := _w4;
_w5 := TRUE AND SerEn_1;
_w6 := ((_w5 AND G_ManMode) AND H_Ax1MovP1PB OR _w5 AND ZAxMovInit_A OR _w5 AND ZAxMovInit1A OR _w5 AND PickModInitA.Y_ZToInit) AND NOT Ax1GoP1;
IF _w6 THEN Ax1AbsPos := Ax1PosP1; END_IF
_w7 := ((_w5 AND G_ManMode) AND H_Ax1MovP2PB OR _w5 AND ZAxMovPick_A) AND O_ModASftC_R AND NOT Ax1GoP2;
IF _w7 THEN Ax1AbsPos := Ax1PosP2; END_IF
_w8 := ((_w5 AND G_ManMode) AND H_Ax1MovP3PB OR _w5 AND ZAxMovPlaceA) AND O_ModASftC_W AND NOT Ax1GoP3;
IF _w8 THEN Ax1AbsPos := Ax1PosP3; END_IF
_w9 := ((_w5 AND G_ManMode) AND H_Ax1MovP1PB OR _w5 AND ZAxMovInit_A OR _w5 AND ZAxMovInit1A OR _w5 AND PickModInitA.Y_ZToInit) AND NOT Ax1GoP1 OR ((_w5 AND G_ManMode) AND H_Ax1MovP2PB OR _w5 AND ZAxMovPick_A) AND O_ModASftC_R AND NOT Ax1GoP2 OR ((_w5 AND G_ManMode) AND H_Ax1MovP3PB OR _w5 AND ZAxMovPlaceA) AND O_ModASftC_W AND NOT Ax1GoP3;
Ax1AbsMove := _w9;

END_PROGRAM
